// TIA Portal V16 export
// export: Created 2024-06-24T15:23:07.0609053Z, ExportSetting WithDefaults, DisplayName Totally Integrated Automation Portal, DisplayVersion V16, DisplayName TIA Portal Version Control Interface, DisplayVersion V16, DisplayName TIA Portal Openness, DisplayVersion V16, DisplayName STEP 7 Professional, DisplayVersion V16, DisplayName STEP 7 Safety, DisplayVersion V16, DisplayName WinCC Advanced, DisplayVersion V16
FUNCTION_BLOCK "FB_Conveyor"   // FB3, LAD
{ S7_Optimized_Access := 'TRUE' }
VERSION : 0.1
// stored: AutoNumber true, IsIECCheckEnabled false, IsRetainMemResEnabled false, MemoryReserve 100, SetENOAutomatically false, UDAEnableTagReadback false
   VAR_INPUT
      "machine ready" : Bool;
      photoeye : Bool;
   END_VAR
   VAR_OUTPUT
      forward : Bool;
      "counter" : Int;
   END_VAR
   VAR_IN_OUT
      start : Bool;
      done : Bool;
   END_VAR
   VAR
      "step" : Array[0..19] of Bool;
   END_VAR
   VAR_TEMP   // added for the SCL form of the ladder/FBD networks
      _w1 : Bool;
   END_VAR
BEGIN

REGION Network 1
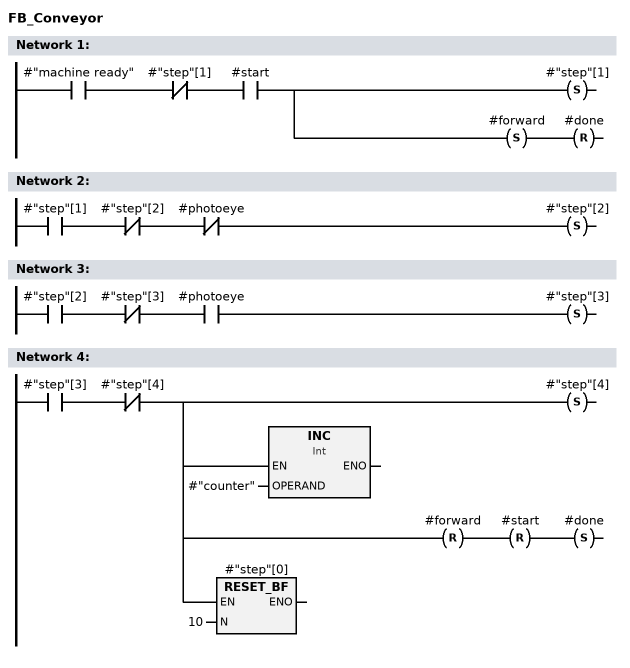
   RUNG wire#powerrail
      Contact( #"machine ready" )
      I_Contact( #"step"[1] )
      Contact( #start )
      wire#w1
      S_Coil( #"step"[1] )
   END_RUNG
   RUNG wire#w1
      S_Coil( #forward )
      R_Coil( #done )
   END_RUNG
   // the same network as SCL:
   #_w1 := #"machine ready" AND NOT #"step"[1] AND #start;
   IF #_w1 THEN
       #"step"[1] := TRUE;
       #forward := TRUE;
       #done := FALSE;
   END_IF;
END_REGION

REGION Network 2
   RUNG wire#powerrail
      Contact( #"step"[1] )
      I_Contact( #"step"[2] )
      I_Contact( #photoeye )
      S_Coil( #"step"[2] )
   END_RUNG
   // the same network as SCL:
   IF #"step"[1] AND NOT #"step"[2] AND NOT #photoeye THEN #"step"[2] := TRUE; END_IF;
END_REGION

REGION Network 3
   RUNG wire#powerrail
      Contact( #"step"[2] )
      I_Contact( #"step"[3] )
      Contact( #photoeye )
      S_Coil( #"step"[3] )
   END_RUNG
   // the same network as SCL:
   IF #"step"[2] AND NOT #"step"[3] AND #photoeye THEN #"step"[3] := TRUE; END_IF;
END_REGION

REGION Network 4
   // no SCL statement known for RBitfield: written as a call
   #_w1 := #"step"[3] AND NOT #"step"[4];
   IF #_w1 THEN
       #"step"[4] := TRUE;
       #"counter" := #"counter" + 1;
       #forward := FALSE;
       #start := FALSE;
       #done := TRUE;
       RESET_BF(operand := #"step"[0], n := 10);
   END_IF;
END_REGION
END_FUNCTION_BLOCK
